// TIA Portal V19 export
TYPE "udt_FlyingCarriage_Parameter"
   STRUCT
      PosTolerance : LReal := 0.1;
      PosWindowDelay : Time := T#100MS;
      ZeroChk_SensorPosition : LReal := 73.17;
      ZeroChk_PosTolerance : LReal := 1.0;
      Limits : Struct
         SwLimNegative : LReal := 0.0;
         SwLimPositive : LReal := 1500.0;
      END_STRUCT;
      Referencing : Struct
         ApprochVelocity : LReal;
         HomingVelocity : LReal;
         HomePositionOffset : LReal;
         HomePosition : LReal;
      END_STRUCT;
      Man : Struct
         Vel : LReal := 5.0;
         Acc : LReal := 5.0;
         Dec : LReal := 5.0;
         Jerk : LReal := 50.0;
      END_STRUCT;
      Aut : Struct
         Vel : LReal := 5.0;
         Acc : LReal := 5.0;
         Dec : LReal := 5.0;
         Jerk : LReal := 50.0;
      END_STRUCT;
      Axis_Kv : LReal := 0.0;
      Drive_Kp : Real := 0.0;
      Drive_Ki : Real := 0.0;
   END_STRUCT;
END_TYPE
